SUBAPPLICATION eio_ueb (* Subapplication Type *)
  (* Standard: 61499-2 *)
  (* Version 1.0, 2025-07-29, franz *)
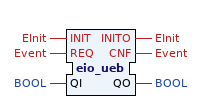
  EVENT_INPUT
    INIT : EInit; (* Initialization Request *)
    REQ; (* Normal Execution Request *)
  END_EVENT
  EVENT_OUTPUT
    INITO : EInit; (* Initialization Confirm *)
    CNF; (* Execution Confirmation *)
  END_EVENT
  VAR_INPUT
    QI : BOOL; (* Input event qualifier *)
  END_VAR
  VAR_OUTPUT
    QO : BOOL; (* Output event qualifier *)
  END_VAR
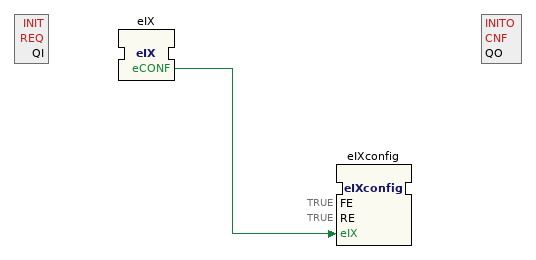
  FBS
    eIX : eIX;
    eIXconfig : eIXconfig(FE := TRUE, RE := TRUE);
  END_FBS
  ADAPTER_CONNECTIONS
    eIX.eCONF TO eIXconfig.eIX;
  END_CONNECTIONS
END_SUBAPPLICATION
